INTERFACE I_DataLogger

METHOD LogCycleData : BOOL
VAR_INPUT
    StationName : STRING(40);
    StepNumber  : INT;
    CycleTimeMs : LREAL;
END_VAR
END_METHOD

METHOD Flush : BOOL
END_METHOD

PROPERTY IsEnabled : BOOL
GET
END_GET
END_PROPERTY

END_INTERFACE

(* stored: Version 1.1.0.1
   Itf I_DataLogger: Id {a86bbf96-76b1-4e91-94ef-4ff83e87e23d}
   Method LogCycleData: Id {eaa38c8d-c6fe-43ff-920a-a531e9c8c2e0}
   Method Flush: Id {28654dbd-a707-46ef-b583-74356eccf678}
   Property IsEnabled: Id {c7345c14-3a2a-4b90-88ee-3459f0797b50}
   Get Get: Id {6713025c-7cec-4fc3-b407-a82aa2fad959} *)
